RoboDK station: Name Engraving Scara Robot.rdk

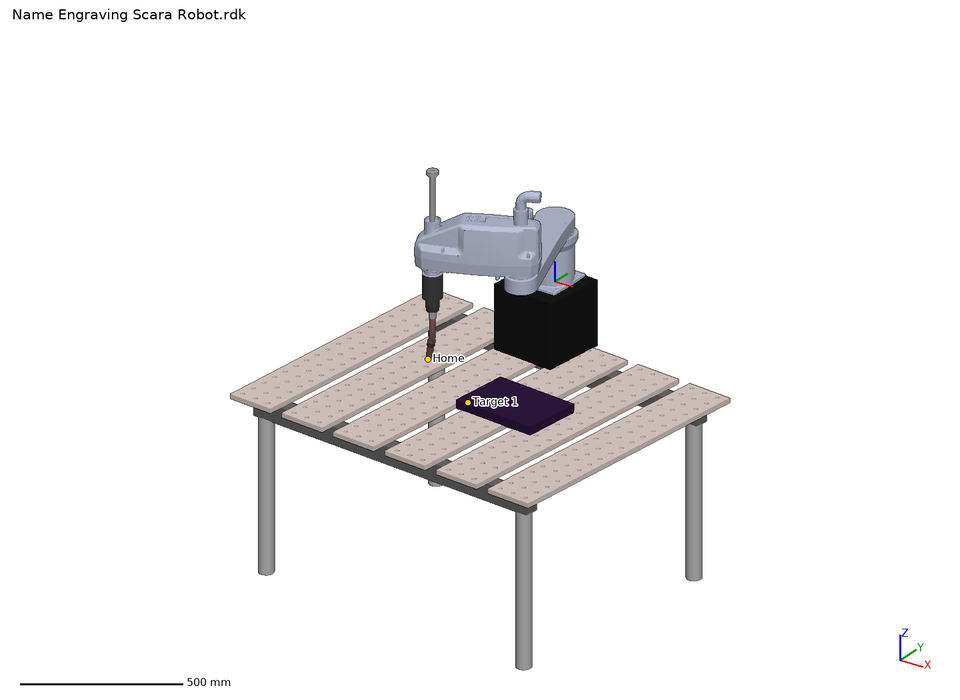
[picture v0: the station drawn from its stored meshes, robots at their saved joint values, targets as dots, program paths as lines]
Station Name Engraving Scara Robot (saved by RoboDK 5.3.0). Poses are relative to the parent item; angles as X-Y-Z fixed-axis rotations.
  - frame Mitsubishi RH-6CH70 Base at (0, 160.3, 0) mm
    - robot Mitsubishi RH-6CH70: 4 axes, payload 6 kg, reach 700 mm, repeatability 0.025 mm, weight 18 kg
        modified DH rows (alpha deg, a mm, theta deg, d mm): 0, 0, 0, 0; 0, 425, 0, 0; 0, 275, 0, -50 linear; 180, 0, 0, 0
        joint limits [-132, -150, 0, -360] to [132, 150, 200, 360]; home [0, 0, 200, 0]; saved at [-69.237, -84.97, 200, 107.177]
      - tool Welding Gun, TCP at (-91, 0, -280) mm, size 122.1 x 64 x 340.8 mm
    - object A4_Platform at (43.61, -515.92, -220.95) mm, rotated rx 0 ry 0 rz -10.11 deg, size 314.2 x 235.1 x 30 mm, geometry from a4_woodenblock.sld
    - target Home (Cartesian target) at (-158.96, -450.47, -130) mm, rotated rx 0 ry 0 rz -47.03 deg; joints [-69.237, -84.97, 200, 107.177] of Mitsubishi RH-6CH70
    - target Target 1 (Cartesian target) at (43.61, -525.92, -190.95) mm, rotated rx 0 ry 0 rz -10.11 deg; joints [-47.577, -76.356, 139.05, 113.822] of Mitsubishi RH-6CH70
  - Python program Prog1 (listed below)
  - object Object Table at (0, 0, 0) mm, size 1193.8 x 965.2 x 609.6 mm, geometry from Object Table.wrl
  - object box at (0, 0, 0) mm, size 225 x 225 x 225 mm, geometry from box.sld

--- Python program Prog1 ---
#A short name engraving program by Muhammad Imran bin Ismael 1810633
from robolink import *    # RoboDK's API
from robodk import *      # Math toolbox for robots
import csv                # To import excel file


# Opening Excel Files
file = open("C:/Users/user/Documents/SEM 1 2122/Robotics/NameCoordinates.csv")
csvreader = csv.reader(file)
header = next(csvreader)
print(header)
rows = []
for row in csvreader:
    rows.append(row)

# Converting the list of list into floats to ease of additions
rows = [list(map(float, sublist)) for sublist in rows]
print(rows) # For verification of floats type

# Start the RoboDK API:
RDK = Robolink()

# Get the robot (first robot found):
robot = RDK.Item('', ITEM_TYPE_ROBOT)

# Get the reference target by name:
target = RDK.Item('Target 1')
home=RDK.Item('Home')
target_pose = target.Pose()
xyz_ref = [target_pose.Pos()]
print(xyz_ref) # For verification of floats type
robot.MoveJ(home) # Move to Home position
robot.MoveJ(target) # Move to Target 1 position


# Start engraving name:MUHAMMAD IMRAN BIN ISMAEL
for i in range(2030): # 2030 as in the number of total coordinates
    # Calculate the new position:
    x = xyz_ref[0][0]+ (rows[i][0]/8)
    y = xyz_ref[0][1]+ (rows[i][1]/8)
    z = xyz_ref[0][2]
    target_pose.setPos([x,y,z])
    robot.MoveL(target_pose)

# Trigger a program call at the end of the movement
robot.RunInstruction('Program_Done')
